FUNCTION_BLOCK FB_Enfield_LSV_PWM_SolenoidControl
VAR_INPUT
END_VAR
VAR_OUTPUT
END_VAR
VAR
	bDigitalIn			AT %I*		: BOOL;
	bReady				AT %I*		: BOOL;
	bHWError			AT %I*		: BOOL;
	bEnableDither		AT %Q*		: BOOL := TRUE;
	bEnable				AT %Q*		: BOOL := TRUE;
	bReset				AT %Q*		: BOOL;
	nPWMOut				AT %Q*		: INT;
END_VAR

//To use call the Enable method to enable the controller 
//Then call the Actuate method to set a duty cycle percentage (100 = Full positive, -100 = Full reverse)

METHOD Actuate : BOOL
VAR_INPUT
	DutyCycle		:INT;
END_VAR
IF bEnable AND bReady THEN
	nPWMOut := DutyCycle * 327;		//Quasi-scale the -100 to 100 percentage input to basic engineering units for the IO terminal doesn't need to be exact in this case
END_IF
END_METHOD

METHOD Disable : BOOL
VAR_INPUT
END_VAR
bEnable := FALSE;
bEnableDither := FALSE;
nPWMOut := 0;
END_METHOD

METHOD Enable : BOOL
VAR_INPUT
END_VAR
bEnable := TRUE;
bEnableDither := TRUE;
END_METHOD

PROPERTY Ready : BOOL
GET
Ready := bReady;
END_GET
END_PROPERTY

{warning 'add method implementation '}
METHOD Reset : BOOL
IF bHWError THEN
	bReset := TRUE;
END_IF
END_METHOD

END_FUNCTION_BLOCK

(* stored: Version 1.1.0.1, ProductVersion 3.1.4024.9
   POU FB_Enfield_LSV_PWM_SolenoidControl: Id {4d3db539-b21d-4626-9305-53445169e987}, SpecialFunc None
   Method Actuate: Id {f7d4aa18-3394-496d-b41d-b6fd90e4462e}
   Method Disable: Id {526a1e03-e255-42d7-9104-15d6642f2fa6}
   Method Enable: Id {91806581-72ee-4587-b970-86928f1db6b1}
   Property Ready: Id {cc025c43-a51d-4a7a-a68a-b0c3a9d58fcb}
   Get Get: Id {43febbc4-5104-43cc-8469-3e2fe70979db}
   Method Reset: Id {58f73db4-6076-4aac-b4ca-18a00cf4695c} *)
